// TIA Portal V17 export
// export: Created 2025-03-07T09:18:38.9601076Z, ExportSetting WithDefaults, DisplayName Totally Integrated Automation Portal, DisplayVersion V17 Update 8, DisplayName TIA Portal Openness, DisplayVersion V17 Update 8, DisplayName TIA Portal Version Control Interface, DisplayVersion V17, DisplayName SINAMICS Startdrive Advanced, DisplayVersion V17 SP2, DisplayName SINAMICS Startdrive G110M, G120, G120C, G120D, G120P, G115D, DisplayVersion V17 SP2, DisplayName SINAMICS Startdrive G130, G150, S120, S150, SINAMICS MV, S210, DisplayVersion V17 SP2, DisplayName STEP 7 Professional, DisplayVersion V17 Update 8, DisplayName SINUMERIK ONE STEP 7 Toolbox, DisplayVersion V17 Update 12, DisplayName SINUMERIK 840D sl STEP 7 Toolbox, DisplayVersion V17 Update 12, DisplayName STEP 7 Safety, DisplayVersion V17 Update 6, DisplayName WinCC Advanced, DisplayVersion V17 Update 8
DATA_BLOCK "DB1018_SAFETY_TAGS"   // DB1018, F_DB
{ S7_Optimized_Access := 'TRUE'; DB_Accessible_From_OPC_UA := 'FALSE' }
AUTHOR : ETXETAR
VERSION : 1.0
// stored: AutoNumber false, DBAccessibleFromOPCUA false, DBAccessibleFromWebserver true
   VAR
      ALWAYS_ON : Bool := TRUE;   // SAFETY ALWAYS ON
      ALWAYS_OFF : Bool;   // SAFETY ALWAYS OFF
      E_STOP_RESET_OPTION : Bool;   // E-STOP RESET OPTION
      SAFETY_GATES_RESET_OPTION : Bool;   // SAFETY GATES RESET OPTION
      PHD_SAFETY_DOOR_OPTION : Bool;   // PART HANDLING DEVICE DOOR OPTION
      AX_NO_INT_EV_ACTIVE : Bool;   // AXES NO INTERNAL EVENT ACTIVE
      SP_NO_INT_EV_ACTIVE : Bool;   // SPINDLES NO INTERNAL EVENT ACTIVE
      AXES_SSM : Bool;   // AXES SSM ACTIVE
      SP_SSM : Bool;   // SPINDLES SSM ACTIVE
      AXES_SOS : Bool;   // AXES SAFETY OPERATING STOP
      SP_SOS : Bool;   // SPINDLES SAFETY OPERATING STOP
      E_STOP_OK : Bool;   // EMERGENCY STOP OK
      E_STOP_OK_OFF_DEL_2 : Bool;   // EMERGENCY STOP OK OFF DELAYED 2
      E_STOP_OK_OFF_DEL_3 : Bool;   // EMERGENCY STOP OK OFF DELAYED 3
      E_STOP_OK_OFF_DEL_4 : Bool;   // EMERGENCY STOP OK OFF DELAYED 4
      E_STOP_RESET : Bool;   // EMERGENCY STOP RESET
      E_STOP_RESET_REQ : Bool;   // EMERGENCY STOP RESET REQUEST
      E_STOP_GANTRY_ROBOT : Bool;   // EMERGENCY STOP GANTRY / EMERGENCY STOP GANTRY-ROBOT
      E_STOP_INPUT : Bool;   // EMERGENCY STOP INPUTS
      MACHINE_E_STOP_OK : Bool;   // EMERGENCY STOP OK / MACHINE EMERGENCY STOP OK
      MACHINE_E_STOP : Bool;   // EMERGENCY STOP OK / MACHINE EMERGENCY STOP
      MACHINE_E_STOP_ALARM : Bool;   // MACHINE EMERGENCY STOP ALARM
      MACHINE_SWITCH_OFF : Bool;   // MACHINE SWITCH OFF
      SAFE_DOORS_U01_CLOSED_AND_LOCKED : Bool;   // MACHINE SAFETY GATES CLOSED AND LOCKED / MACHINE SAFETY DOORS CLOSED AND LOCKED
      SAFE_DOORS_U01_CLOSED_AND_LOCKED_OFF_DEL_2 : Bool;   // MACHINE SAFETY GATES CLOSED AND LOCKED OFF DELAYED 2 / MACHINE SAFETY DOORS CLOSED AND LOCKED OFF DELAYED 2
      SAFE_DOORS_U01_CLOSED_AND_LOCKED_OFF_DEL_3 : Bool;   // MACHINE SAFETY GATES CLOSED AND LOCKED OFF DELAYED 3 / MACHINE SAFETY DOORS CLOSED AND LOCKED OFF DELAYED 3
      SAFE_DOORS_U01_CLOSED_AND_LOCKED_OFF_DEL_4 : Bool;   // MACHINE SAFETY GATES CLOSED AND LOCKED OFF DELAYED 4 / MACHINE SAFETY DOORS CLOSED AND LOCKED OFF DELAYED 4
      SAFE_DOORS_CLOSED_AND_LOCKED_RESET : Bool;   // MACHINE SAFETY GATES CLOSED AND LOCKED RESET / MACHINE SAFETY DOORS CLOSED AND LOCKED RESET
      SAFE_DOORS_CLOSED_AND_LOCKED_RESET_REQ : Bool;   // MACHINE SAFETY GATES CLOSED AND LOCKED RESET REQUEST / MACHINE SAFETY DOORS CLOSED AND LOCKED RESET REQUEST
      SAFE_DOORS_CLOSED_AND_LOCKED_FOR_GANTRY_ROBOT : Bool;   // LOAD/UNLOAD + PART HANDLING DEVICE SAFETY DOORS CLOSED AND LOCKED / SAFETY DOORS CLOSED AND LOCKED FOR GANTRY-ROBOT
      SAFE_DOORS_U02_CLOSED_AND_LOCKED : Bool;   // MACHINE SAFETY GATES CLOSED AND LOCKED / MACHINE SAFETY DOORS CLOSED AND LOCKED
      SAFE_DOORS_U02_CLOSED_AND_LOCKED_OFF_DEL_2 : Bool;   // MACHINE SAFETY GATES CLOSED AND LOCKED OFF DELAYED 2 / MACHINE SAFETY DOORS CLOSED AND LOCKED OFF DELAYED 2
      SAFE_DOORS_U02_CLOSED_AND_LOCKED_OFF_DEL_3 : Bool;   // MACHINE SAFETY GATES CLOSED AND LOCKED OFF DELAYED 3 / MACHINE SAFETY DOORS CLOSED AND LOCKED OFF DELAYED 3
      SAFE_DOORS_U02_CLOSED_AND_LOCKED_OFF_DEL_4 : Bool;   // MACHINE SAFETY GATES CLOSED AND LOCKED OFF DELAYED 4 / MACHINE SAFETY DOORS CLOSED AND LOCKED OFF DELAYED 4
      FEEDBACK_OFF_CLS_LCKD_GANTRY_ROBOT : Bool;   // FEEDBACK OFF SAFETY DOORS CLOSED AND LOCKED FOR GANTRY-ROBOT
      FEEDBACK_OFF_CLS_LCKD_GANTRY_ROBOT_ALARM : Bool;   // FEEDBACK OFF SAFETY DOORS CLOSED AND LOCKED FOR GANTRY-ROBOT ALARM
      POWER_ON_W_ENABLE_BUTT : Bool;   // POWER ON WITH HT8 ENABLE BUTTON / POWER ON WITH HT10 ENABLE BUTTON
      POWER_ON_W_ENABLE_BUTT_OFF_DEL_2 : Bool;   // POWER ON WITH HT8 ENABLE BUTTON OFF DELAYED 2 / POWER ON WITH HT10 ENABLE BUTTON OFF DELAYED 2
      POWER_ON_W_ENABLE_BUTT_OFF_DEL_3 : Bool;   // POWER ON WITH HT8 ENABLE BUTTON OFF DELAYED 3 / POWER ON WITH HT10 ENABLE BUTTON OFF DELAYED 3
      POWER_ON_W_ENABLE_BUTT_OFF_DEL_4 : Bool;   // POWER ON WITH HT8 ENABLE BUTTON OFF DELAYED 4 / POWER ON WITH HT10 ENABLE BUTTON OFF DELAYED 4
      POWER_ON_W_ENABLE_BUTT_RESET : Bool;   // POWER ON WITH HT8 ENABLE BUTTON RESET / POWER ON WITH HT10 ENABLE BUTTON RESET
      POWER_ON_W_ENABLE_BUTT_RESET_REQ : Bool;   // POWER ON WITH HT8 ENABLE BUTTON RESET REQUEST / POWER ON WITH HT10 ENABLE BUTTON RESET REQUEST
      POWER_ON_W_ENABLE_OUT : Bool;   // POWER ON WITH HT10 ENABLE BUTTON OUTPUT
      FEEDBACK_OFF_POWER_ENABLE : Bool;   // FEEDBACK OFF POWER ENABLE
      FEEDBACK_OFF_POWER_ENABLE_ALARM : Bool;   // FEEDBACK OFF POWER ENABLE ALARM
      ENABLING_DEV_SWTCHD_ON_FROM_UNIT_01_STATION_02_DOOR_AREA : Bool;   // MACHININIG SAFETY DOOR OPENED AND ENABLING DEVICE SWITCHED ON / UNIT 01 STATION 02 SAFETY DOOR OPENED AND ENABLING DEVICE SWITCHED ON
      ENABLING_DEV_SWTCHD_ON_FROM_UNIT_01_MAIN_SAFETY_DOOR_AREA : Bool;   // MACHININIG SAFETY DOOR OPENED AND ENABLING DEVICE SWITCHED ON / UNIT 01 MAIN SAFETY SAFETY DOOR OPENED AND ENABLING DEVICE SWITCHED ON
      ENABLING_DEV_SWTCHD_ON_FROM_UNIT_01_STATION_04_DOOR_AREA : Bool;   // MAGAZINE SAFETY DOOR OPENED AND ENABLING DEVICE SWITCHED ON / UNIT 01 STATION 04 SAFETY DOOR OPENED AND ENABLING DEVICE SWITCHED ON
      ENABLING_DEV_SWTCHD_ON_FROM_UNIT_01_MAINTENANCE_DOOR_AREA : Bool;   // MAGAZINE SAFETY DOOR OPENED AND ENABLING DEVICE SWITCHED ON / UNIT 01 MAINTENANCE SAFETY DOOR OPENED AND ENABLING DEVICE SWITCHED ON
      ENABLING_DEV_SWTCHD_ON_FROM_UNIT_02_STATION_02_DOOR_AREA : Bool;   // MAGAZINE SAFETY DOOR OPENED AND ENABLING DEVICE SWITCHED ON / UNIT 02 STATION 02 SAFETY DOOR OPENED AND ENABLING DEVICE SWITCHED ON
      ENABLING_DEV_SWTCHD_ON_FROM_UNIT_02_MAIN_SAFETY_DOOR_AREA : Bool;   // MAGAZINE SAFETY DOOR OPENED AND ENABLING DEVICE SWITCHED ON / UNIT 02 MAIN SAFETY DOOR OPENED AND ENABLING DEVICE SWITCHED ON
      ENABLING_DEV_SWTCHD_ON_FROM_UNIT_02_STATION_04_DOOR_AREA : Bool;   // LOAD/UNLOAD SAFETY DOOR OPENED AND ENABLING DEVICE SWITCHED ON / UNIT 02 STATION 04 SAFETY DOOR OPENED AND ENABLING DEVICE SWITCHED ON
      ENABLING_DEV_SWTCHD_ON_FROM_UNIT_02_MAINTENANCE_DOOR_AREA : Bool;   // PART HANDLING DEVICE SAFETY DOOR OPENED AND ENABLING DEVICE SWITCHED ON / UNIT 02 MAINTENANCE SAFETY DOOR OPENED AND ENABLING DEVICE SWITCHED ON
      ENABLING_DEV_SWTCHD_ON_FROM_ROBOT_CELL_DOOR_AREA : Bool;   // ROBOT CELL SAFETY DOOR OPENED AND ENABLING DEVICE SWITCHED ON
      MACHINE_BA1_MODE_SELECTED : Bool;   // MACHINE BA1 MODE SELECTED
      MACHINE_BA2_MODE_SELECTED : Bool;   // MACHINE BA2 MODE SELECTED
      MACHINE_BA3_MODE_SELECTED : Bool;   // MACHINE BA3 MODE SELECTED
      ENABLE_DEVICE_FROM_UNIT_01_STATION_02_DOOR_AREA : Bool;   // ENABLE DEVICE FROM MACHINING DOOR AREA / ENABLE DEVICE FROM UNIT 01 STATION 02 DOOR AREA
      ENABLE_DEVICE_FROM_UNIT_01_MAIN_SAFETY_DOOR_AREA : Bool;   // ENABLE DEVICE FROM MACHINING DOOR AREA / ENABLE DEVICE FROM UNIT 01 MAIN SAFETY DOOR AREA
      ENABLE_DEVICE_FROM_UNIT_01_STATION_04_DOOR_AREA : Bool;   // ENABLE DEVICE FROM MAGAZINE DOOR AREA / ENABLE DEVICE FROM UNIT 01 STATION 04 DOOR AREA
      ENABLE_DEVICE_FROM_UNIT_01_MAINTENANCE_DOOR_AREA : Bool;   // ENABLE DEVICE FROM MAGAZINE DOOR AREA / ENABLE DEVICE FROM UNIT 01 MAINTENANCE DOOR AREA
      ENABLE_DEVICE_FROM_UNIT_02_STATION_02_DOOR_AREA : Bool;   // ENABLE DEVICE FROM MAGAZINE DOOR AREA / ENABLE DEVICE FROM UNIT 02 STATION 02 DOOR AREA
      ENABLE_DEVICE_FROM_UNIT_02_MAIN_SAFETY_DOOR_AREA : Bool;   // ENABLE DEVICE FROM MAGAZINE DOOR AREA / ENABLE DEVICE FROM UNIT 02 MAIN DOOR AREA
      ENABLE_DEVICE_FROM_UNIT_02_STATION_04_DOOR_AREA : Bool;   // ENABLE DEVICE FROM LOAD/UNLOAD DOOR AREA / ENABLE DEVICE FROM UNIT 02 STATION 04 DOOR AREA
      ENABLE_DEVICE_FROM_UNIT_02_MAINTENANCE_DOOR_AREA : Bool;   // ENABLE DEVICE FROM PART HANDLING DEVICE DOOR AREA / ENABLE DEVICE FROM UNIT 02 MAINTENANCE DOOR AREA
      ENABLE_DEVICE_FROM_ROBOR_CELL_DOOR_AREA : Bool;   // ENABLE DEVICE FROM ROBOT CELL DOOR AREA
      MACHINE_IN_MANUAL_MODE : Bool;   // MACHINE IN MANUAL MODE
      RESET_FAULTS : Bool;   // RESET FAULTS
      ENABLE_BUTTON_PRESED_RESET_SI_RELAY : Bool;   // ENABLE BUTTON PRESED RESET SI RELAY
      DESELECT_SPINDLE_STO_01R : Bool;   // DESELECT SPINDLE STO 01R
      DESELECT_SPINDLE_STO_01L : Bool;   // DESELECT SPINDLE STO 01L
      ALL_AC_MOTORS_OFF_SWITCHED : Bool;   // ALL AC MOTORS OFF SWITCHED
      MACHINE_SWITCH_OFF_1 : Bool;   // MACHINE SWITCH OFF 1
      HT10_CONNECTED_TO_MACHINE_MAIN_PANEL : Bool;   // HT10 CONNECTED TO MACHINE MAIN PANEL
      HT10_CONNECTED_TO_TOOL_MAGAZINE_AREA_CONNECTION_BOX : Bool;   // HT10 CONNECTED TO MAGAZINE AREA CONNECTION BOX
      HT10_CONNECTED_TO_LOAD_UNLOAD_DOOR_AREA : Bool;   // HT10 CONNECTED TO LOAD UNLOAD DOOR AREA
      COOLANT_OFF_01R_SET_SPINDLES_SBH_SLS : Bool;   // COOLANT OFF 01R (SET SPINDLES SBH-SG)
      COOLANT_OFF_01L_SET_SPINDLES_SBH_SLS : Bool;   // COOLANT OFF 01L (SET SPINDLES SBH-SG)
      MANUAL_LOAD_SELECTED : Bool;   // MANUAL LOAD SELECTED
      MANUAL_LOAD_PHD_SAFETY_DOOR : Bool;   // MANUAL LOAD - PHD SAFETY DOOR
      "E-STOP_FEEDBACK_OFF_OK" : Bool;   // E-STOP FEEDBACK OFF OK
      MACHINE_SAFETY_DOOR_FEEDBACK_OFF_OK : Bool;   // MACHINE SAFETY DOOR FEEDBACK OFF OK
      LOAD_UNLOAD_SAFETY_DOOR_FEEDBACK_OFF_OK : Bool;   // LOAD UNLOAD SAFETY DOOR FEEDBACK OFF OK
      POWER_ENABLE_FEEDBACK_OFF_OK : Bool;   // POWER ENABLE FEEDBACK OFF OK
      LASER_SOURCE_ENABLE_CONDITIONS : Bool;   // POWER ON WITH HT8 ENABLE BUTTON / LASER SOURCE ENABLE CONDITIONS
      FEEDBACK_OFF_LASER_SOURCE_ENABLE_CONDITIONS : Bool;   // FEEDBACK OFF LASER SOURCE ENABLE CONDITIONS
      FEEDBACK_OFF_LASER_SOURCE_ENABLE_CONDITIONS_ALARM : Bool;   // FEEDBACK OFF LASER SOURCE ENABLE CONDITIONS ALARM
      MANUAL_LOAD_CLOSE_AUTO_DOOR_BIMANUAL : Bool;   // MANUAL LOAD MODE CLOSE AUTOMATIC DOOR WITH BIMANUAL
      MANUAL_LOAD_OPEN_AUTO_DOOR_WO_BIMANUAL : Bool;   // MANUAL LOAD MODE OPEN AUTOMATIC DOOR WITHOUT BIMANUAL
      GROUP_1_E10 : "SAFETY_GROUP";   // GROUP 1 (E10)
      GROUP_2_C11_Z11 : "SAFETY_GROUP";   // GROUP 2 (C11)
      GROUP_3_C12 : "SAFETY_GROUP";   // GROUP 3 (C12)
      GROUP_4_C13_X13_Z13 : "SAFETY_GROUP";   // GROUP 4 (C13-X13-Z13)
      GROUP_5_C14_Z14 : "SAFETY_GROUP";   // GROUP 5 (C14)
      GROUP_6_E20 : "SAFETY_GROUP";   // GROUP 6 (E20)
      GROUP_7_C21_Z21 : "SAFETY_GROUP";   // GROUP 7 (C21)
      GROUP_8_C22 : "SAFETY_GROUP";   // GROUP 8 (C22)
      GROUP_9_C23_X23_Z23 : "SAFETY_GROUP";   // GROUP 9 (C23-X23-Z23)
      GROUP_10_C24_Z24 : "SAFETY_GROUP";   // GROUP 10 (C24)
      GROUP_11_X31 : "SAFETY_GROUP";   // GROUP 11 (Xc-Yc-Zc)
      POWDER_E_STOP_OK : Bool;   // POWDER ZONE EMERGENCY STOP OK
      POWDER_SAFE_DOORS_CLOSED_AND_LOCKED : Bool;   // MACHINE SAFETY GATES CLOSED AND LOCKED / POWDER ZONE SAFETY DOORS CLOSED AND LOCKED
      CELL_E_STOP_OK : Bool;   // ROBOT CELL EMERGENCY STOP OK
      CELL_SAFE_DOORS_CLOSED_AND_LOCKED : Bool;   // MACHINE SAFETY GATES CLOSED AND LOCKED / ROBOT CELL SAFETY DOORS CLOSED AND LOCKED
      ROBOT_OUT_OF_COLLISION_MACHINE_UNIT_01 : Bool;   // ROBOT CELL OUT OF COLLISION MACHINE UNIT 01
      ROBOT_OUT_OF_COLLISION_MACHINE_UNIT_02 : Bool;   // ROBOT CELL OUT OF COLLISION MACHINE UNIT 02
   END_VAR
BEGIN
   // GROUP_1_E10.STO_Deactivate : GROUP 1 SAFE TORQUE OFF DEACTIVATE
   // GROUP_1_E10.SS1_Deactivate : GROUP 1 SAFE STOP 1 DEACTIVATE
   // GROUP_1_E10.SS2_Deactivate : GROUP 1 SAFE STOP 2 DEACTIVATE
   // GROUP_1_E10.SS2E_Deactivate : GROUP 1 SAFE STOP 2 EXTENDED DEACTIVATE
   // GROUP_1_E10.SOS_Deactivate : GROUP 1 SAFE OPERATING STOP DEACTIVATE
   // GROUP_1_E10.SLS_Deactivate : GROUP 1 SAFE LIMITED SPEED DEACTIVATE
   // GROUP_1_E10.SLS_BIT0 : GROUP 1 SAFE LIMITED SPEED BIT 0
   // GROUP_1_E10.SLS_BIT1 : GROUP 1 SAFE LIMITED SPEED BIT 1
   // GROUP_2_C11_Z11.STO_Deactivate : GROUP 2 SAFE TORQUE OFF DEACTIVATE
   // GROUP_2_C11_Z11.SS1_Deactivate : GROUP 2 SAFE STOP 1 DEACTIVATE
   // GROUP_2_C11_Z11.SS2_Deactivate : GROUP 2 SAFE STOP 2 DEACTIVATE
   // GROUP_2_C11_Z11.SS2E_Deactivate : GROUP 2 SAFE STOP 2 EXTENDED DEACTIVATE
   // GROUP_2_C11_Z11.SOS_Deactivate : GROUP 2 SAFE OPERATING STOP DEACTIVATE
   // GROUP_2_C11_Z11.SLS_Deactivate : GROUP 2 SAFE LIMITED SPEED DEACTIVATE
   // GROUP_2_C11_Z11.SLS_BIT0 : GROUP 2 SAFE LIMITED SPEED BIT 0
   // GROUP_2_C11_Z11.SLS_BIT1 : GROUP 2 SAFE LIMITED SPEED BIT 1
   // GROUP_3_C12.STO_Deactivate : GROUP 3 SAFE TORQUE OFF DEACTIVATE
   // GROUP_3_C12.SS1_Deactivate : GROUP 3 SAFE STOP 1 DEACTIVATE
   // GROUP_3_C12.SS2_Deactivate : GROUP 3 SAFE STOP 2 DEACTIVATE
   // GROUP_3_C12.SS2E_Deactivate : GROUP 3 SAFE STOP 2 EXTENDED DEACTIVATE
   // GROUP_3_C12.SOS_Deactivate : GROUP 3 SAFE OPERATING STOP DEACTIVATE
   // GROUP_3_C12.SLS_Deactivate : GROUP 3 SAFE LIMITED SPEED DEACTIVATE
   // GROUP_3_C12.SLS_BIT0 : GROUP 3 SAFE LIMITED SPEED BIT 0
   // GROUP_3_C12.SLS_BIT1 : GROUP 3 SAFE LIMITED SPEED BIT 1
   // GROUP_4_C13_X13_Z13.STO_Deactivate : GROUP 4 SAFE TORQUE OFF DEACTIVATE
   // GROUP_4_C13_X13_Z13.SS1_Deactivate : GROUP 4 SAFE STOP 1 DEACTIVATE
   // GROUP_4_C13_X13_Z13.SS2_Deactivate : GROUP 4 SAFE STOP 2 DEACTIVATE
   // GROUP_4_C13_X13_Z13.SS2E_Deactivate : GROUP 4 SAFE STOP 2 EXTENDED DEACTIVATE
   // GROUP_4_C13_X13_Z13.SOS_Deactivate : GROUP 4 SAFE OPERATING STOP DEACTIVATE
   // GROUP_4_C13_X13_Z13.SLS_Deactivate : GROUP 4 SAFE LIMITED SPEED DEACTIVATE
   // GROUP_4_C13_X13_Z13.SLS_BIT0 : GROUP 4 SAFE LIMITED SPEED BIT 0
   // GROUP_4_C13_X13_Z13.SLS_BIT1 : GROUP 4 SAFE LIMITED SPEED BIT 1
   // GROUP_5_C14_Z14.STO_Deactivate : GROUP 5 SAFE TORQUE OFF DEACTIVATE
   // GROUP_5_C14_Z14.SS1_Deactivate : GROUP 5 SAFE STOP 1 DEACTIVATE
   // GROUP_5_C14_Z14.SS2_Deactivate : GROUP 5 SAFE STOP 2 DEACTIVATE
   // GROUP_5_C14_Z14.SS2E_Deactivate : GROUP 5 SAFE STOP 2 EXTENDED DEACTIVATE
   // GROUP_5_C14_Z14.SOS_Deactivate : GROUP 5 SAFE OPERATING STOP DEACTIVATE
   // GROUP_5_C14_Z14.SLS_Deactivate : GROUP 5 SAFE LIMITED SPEED DEACTIVATE
   // GROUP_5_C14_Z14.SLS_BIT0 : GROUP 5 SAFE LIMITED SPEED BIT 0
   // GROUP_5_C14_Z14.SLS_BIT1 : GROUP 5 SAFE LIMITED SPEED BIT 1
   // GROUP_6_E20.STO_Deactivate : GROUP 6 SAFE TORQUE OFF DEACTIVATE
   // GROUP_6_E20.SS1_Deactivate : GROUP 6 SAFE STOP 1 DEACTIVATE
   // GROUP_6_E20.SS2_Deactivate : GROUP 6 SAFE STOP 2 DEACTIVATE
   // GROUP_6_E20.SS2E_Deactivate : GROUP 6 SAFE STOP 2 EXTENDED DEACTIVATE
   // GROUP_6_E20.SOS_Deactivate : GROUP 6 SAFE OPERATING STOP DEACTIVATE
   // GROUP_6_E20.SLS_Deactivate : GROUP 6 SAFE LIMITED SPEED DEACTIVATE
   // GROUP_6_E20.SLS_BIT0 : GROUP 6 SAFE LIMITED SPEED BIT 0
   // GROUP_6_E20.SLS_BIT1 : GROUP 6 SAFE LIMITED SPEED BIT 1
   // GROUP_7_C21_Z21.STO_Deactivate : GROUP 7 SAFE TORQUE OFF DEACTIVATE
   // GROUP_7_C21_Z21.SS1_Deactivate : GROUP 7 SAFE STOP 1 DEACTIVATE
   // GROUP_7_C21_Z21.SS2_Deactivate : GROUP 7 SAFE STOP 2 DEACTIVATE
   // GROUP_7_C21_Z21.SS2E_Deactivate : GROUP 7 SAFE STOP 2 EXTENDED DEACTIVATE
   // GROUP_7_C21_Z21.SOS_Deactivate : GROUP 7 SAFE OPERATING STOP DEACTIVATE
   // GROUP_7_C21_Z21.SLS_Deactivate : GROUP 7 SAFE LIMITED SPEED DEACTIVATE
   // GROUP_7_C21_Z21.SLS_BIT0 : GROUP 7 SAFE LIMITED SPEED BIT 0
   // GROUP_7_C21_Z21.SLS_BIT1 : GROUP 7 SAFE LIMITED SPEED BIT 1
   // GROUP_8_C22.STO_Deactivate : GROUP 8 SAFE TORQUE OFF DEACTIVATE
   // GROUP_8_C22.SS1_Deactivate : GROUP 8 SAFE STOP 1 DEACTIVATE
   // GROUP_8_C22.SS2_Deactivate : GROUP 8 SAFE STOP 2 DEACTIVATE
   // GROUP_8_C22.SS2E_Deactivate : GROUP 8 SAFE STOP 2 EXTENDED DEACTIVATE
   // GROUP_8_C22.SOS_Deactivate : GROUP 8 SAFE OPERATING STOP DEACTIVATE
   // GROUP_8_C22.SLS_Deactivate : GROUP 8 SAFE LIMITED SPEED DEACTIVATE
   // GROUP_8_C22.SLS_BIT0 : GROUP 8 SAFE LIMITED SPEED BIT 0
   // GROUP_8_C22.SLS_BIT1 : GROUP 8 SAFE LIMITED SPEED BIT 1
   // GROUP_9_C23_X23_Z23.STO_Deactivate : GROUP 8 SAFE TORQUE OFF DEACTIVATE
   // GROUP_9_C23_X23_Z23.SS1_Deactivate : GROUP 8 SAFE STOP 1 DEACTIVATE
   // GROUP_9_C23_X23_Z23.SS2_Deactivate : GROUP 8 SAFE STOP 2 DEACTIVATE
   // GROUP_9_C23_X23_Z23.SS2E_Deactivate : GROUP 8 SAFE STOP 2 EXTENDED DEACTIVATE
   // GROUP_9_C23_X23_Z23.SOS_Deactivate : GROUP 8 SAFE OPERATING STOP DEACTIVATE
   // GROUP_9_C23_X23_Z23.SLS_Deactivate : GROUP 8 SAFE LIMITED SPEED DEACTIVATE
   // GROUP_9_C23_X23_Z23.SLS_BIT0 : GROUP 8 SAFE LIMITED SPEED BIT 0
   // GROUP_9_C23_X23_Z23.SLS_BIT1 : GROUP 8 SAFE LIMITED SPEED BIT 1
   // GROUP_10_C24_Z24.STO_Deactivate : GROUP 8 SAFE TORQUE OFF DEACTIVATE
   // GROUP_10_C24_Z24.SS1_Deactivate : GROUP 8 SAFE STOP 1 DEACTIVATE
   // GROUP_10_C24_Z24.SS2_Deactivate : GROUP 8 SAFE STOP 2 DEACTIVATE
   // GROUP_10_C24_Z24.SS2E_Deactivate : GROUP 8 SAFE STOP 2 EXTENDED DEACTIVATE
   // GROUP_10_C24_Z24.SOS_Deactivate : GROUP 8 SAFE OPERATING STOP DEACTIVATE
   // GROUP_10_C24_Z24.SLS_Deactivate : GROUP 8 SAFE LIMITED SPEED DEACTIVATE
   // GROUP_10_C24_Z24.SLS_BIT0 : GROUP 8 SAFE LIMITED SPEED BIT 0
   // GROUP_10_C24_Z24.SLS_BIT1 : GROUP 8 SAFE LIMITED SPEED BIT 1
   // GROUP_11_X31.STO_Deactivate : GROUP 8 SAFE TORQUE OFF DEACTIVATE
   // GROUP_11_X31.SS1_Deactivate : GROUP 8 SAFE STOP 1 DEACTIVATE
   // GROUP_11_X31.SS2_Deactivate : GROUP 8 SAFE STOP 2 DEACTIVATE
   // GROUP_11_X31.SS2E_Deactivate : GROUP 8 SAFE STOP 2 EXTENDED DEACTIVATE
   // GROUP_11_X31.SOS_Deactivate : GROUP 8 SAFE OPERATING STOP DEACTIVATE
   // GROUP_11_X31.SLS_Deactivate : GROUP 8 SAFE LIMITED SPEED DEACTIVATE
   // GROUP_11_X31.SLS_BIT0 : GROUP 8 SAFE LIMITED SPEED BIT 0
   // GROUP_11_X31.SLS_BIT1 : GROUP 8 SAFE LIMITED SPEED BIT 1
END_DATA_BLOCK
